Fanuc KAREL source: CA0121.KL

-- PROVISIONAL review KL for V940-1; original PC SHA256 a0212965cf7ec0234d3a6533aab3b798ea069698b484b94f20207c0c5d4ccaa1
-- Incomplete behavior may be omitted. Consult companion uncertainty JSON. Do not deploy.
PROGRAM CA0121
%NOLOCKGROUP
BEGIN
  -- V9_ZERO_TABLE_METADATA_HINT layout=0001; no indexed target words; source/name/runtime held
  -- UNRESOLVED_PC offsets 0-1; opcodes 7B
  -- UNRESOLVED_PC offsets 6-20; opcodes 21,9D,52,23
  -- UNRESOLVED_PC offsets 25-42; opcodes 2D,21,52,7F
  -- UNRESOLVED_PC offsets 47-52; opcodes 7F,7B
  -- UNRESOLVED_PC offsets 57-75; opcodes 21,2E,52,23
  -- UNRESOLVED_PC offsets 80-97; opcodes 2D,21,52,7F
  -- UNRESOLVED_PC offsets 102-107; opcodes 7F,7B
  -- UNRESOLVED_PC offsets 112-130; opcodes 21,2E,52,23
  -- UNRESOLVED_PC offsets 135-152; opcodes 2D,21,52,7F
  -- UNRESOLVED_PC offsets 157-162; opcodes 7F,7B
  -- UNRESOLVED_PC offsets 167-181; opcodes 21,9D,52,23
  -- UNRESOLVED_PC offsets 186-190; opcodes 7F
  -- UNRESOLVED_PC offsets 195-202; opcodes 9C,23
  -- UNRESOLVED_PC offsets 207-214; opcodes 9D,23
  -- UNRESOLVED_PC offsets 219-230; opcodes 2E,23
  -- UNRESOLVED_PC offsets 235-242; opcodes 9D,23
  -- UNRESOLVED_PC offsets 247-256; opcodes 3F,75
  -- UNRESOLVED_PC offsets 261-275; opcodes 2E,22,9D,33,35
  -- UNRESOLVED_PC offsets 280-294; opcodes 2E,22,9D,33,35
  -- UNRESOLVED_PC offsets 299-314; opcodes 2E,22,32,35
  -- UNRESOLVED_PC offsets 319-334; opcodes 2E,22,32,35
  -- UNRESOLVED_PC offsets 339-376; opcodes 27,27,27,22,AA,27,27,22,AA,27,27,22,AA,AA
  -- UNRESOLVED_PC offsets 381-385; opcodes 7F
END CA0121
